FUNCTION_BLOCK CylControlILChanOL (* Composite Function Block Type *)
  (* Standard: 61499-2 *)
  (* Version 0.0, 12/6/2023, vaatmar1, nxtControl GmBH, template *)
  PACKAGE Main;
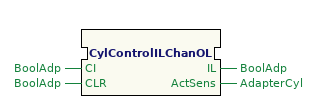
  SOCKETS
    CI : BoolAdp;
    CLR : BoolAdp;
  END_SOCKETS
  PLUGS
    IL : BoolAdp;
    ActSens : AdapterCyl;
  END_PLUGS
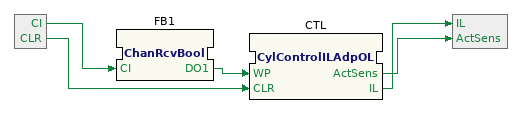
  FBS
    CTL : CylControlILAdpOL;
    FB1 : ChanRcvBool;
  END_FBS
  ADAPTER_CONNECTIONS
    CTL.ActSens TO ActSens;
    CLR TO CTL.CLR;
    CTL.IL TO IL;
    CI TO FB1.CI;
    FB1.DO1 TO CTL.WP;
  END_CONNECTIONS
END_FUNCTION_BLOCK
